LIN {X 0,Y 304.898,Z 957.801,A -85,B 0,C 180,E1 6290.222,E2 6290.222} C_VEL
LIN {X 0,Y 292.236,Z 978.047,A -85,B 0,C 180,E1 6289.106,E2 6289.106} C_VEL
LIN {X 0,Y 278.301,Z 997.321,A -85,B 0,C 180,E1 6287.757,E2 6287.757} C_VEL
LIN {X 0,Y 264.527,Z 1014.363,A -85,B 0,C 180,E1 6286.275,E2 6286.275} C_VEL
LIN {X 0,Y 248.242,Z 1032.202,A -85,B 0,C 180,E1 6284.295,E2 6284.295} C_VEL
LIN {X 0,Y 233.158,Z 1046.985,A -85,B 0,C 180,E1 6282.185,E2 6282.185} C_VEL
LIN {X 0,Y 215.006,Z 1062.935,A -85,B 0,C 180,E1 6279.19,E2 6279.19} C_VEL
LIN {X 0,Y 199.139,Z 1075.414,A -85,B 0,C 180,E1 6276.041,E2 6276.041} C_VEL
LIN {X 0,Y 181.496,Z 1088.037,A -85,B 0,C 180,E1 6271.719,E2 6271.719} C_VEL
LIN {X 0,Y 165.933,Z 1098.063,A -85,B 0,C 180,E1 6266.888,E2 6266.888} C_VEL
LIN {X 0,Y 150.317,Z 1107.482,A -85,B 0,C 180,E1 6260.5,E2 6260.5} C_VEL
LIN {X 0,Y 136.741,Z 1114.997,A -85,B 0,C 180,E1 6252.847,E2 6252.847} C_VEL
LIN {X 0,Y 125.803,Z 1121.052,A -85,B 0,C 180,E1 6243.805,E2 6243.805} C_VEL
LIN {X 0,Y 117.737,Z 1125.633,A -85,B 0,C 180,E1 6232.996,E2 6232.996} C_VEL
LIN {X 0,Y 113.836,Z 1128.278,A -85,B 0,C 180,E1 6223.201,E2 6223.201} C_VEL
LIN {X 0,Y 112.36,Z 1129.83,A -85,B 0,C 180,E1 6213.571,E2 6213.571} C_VEL
LIN {X 0,Y 112.173,Z 1130.41,A -85,B 0,C 180,E1 6205.399,E2 6205.399} C_VEL
LIN {X 0,Y 112.752,Z 1130.33,A -85,B 0,C 180,E1 6196.669,E2 6196.669} C_VEL
LIN {X 0,Y 116.015,Z 1129.028,A -85,B 0,C 180,E1 6184.819,E2 6184.819} C_VEL
LIN {X 0,Y 122.657,Z 1126.25,A -85,B 0,C 180,E1 6174.06,E2 6174.06} C_VEL
LIN {X 0,Y 132.853,Z 1122.064,A -85,B 0,C 180,E1 6164.357,E2 6164.357} C_VEL
LIN {X 0,Y 146.642,Z 1115.907,A -85,B 0,C 180,E1 6155.766,E2 6155.766} C_VEL
LIN {X 0,Y 161.55,Z 1108.77,A -85,B 0,C 180,E1 6149.226,E2 6149.226} C_VEL
LIN {X 0,Y 179.686,Z 1099.063,A -85,B 0,C 180,E1 6143.34,E2 6143.34} C_VEL
LIN {X 0,Y 195.959,Z 1089.416,A -85,B 0,C 180,E1 6139.269,E2 6139.269} C_VEL
LIN {X 0,Y 215.67,Z 1076.309,A -85,B 0,C 180,E1 6135.348,E2 6135.348} C_VEL
LIN {X 0,Y 231.93,Z 1064.205,A -85,B 0,C 180,E1 6132.701,E2 6132.701} C_VEL
LIN {X 0,Y 251.017,Z 1048.279,A -85,B 0,C 180,E1 6130.094,E2 6130.094} C_VEL
LIN {X 0,Y 266.738,Z 1033.492,A -85,B 0,C 180,E1 6128.258,E2 6128.258} C_VEL
LIN {X 0,Y 283.805,Z 1015.52,A -85,B 0,C 180,E1 6126.518,E2 6126.518} C_VEL
LIN {X 0,Y 298.201,Z 998.272,A -85,B 0,C 180,E1 6125.209,E2 6125.209} C_VEL
LIN {X 0,Y 312.738,Z 978.752,A -85,B 0,C 180,E1 6124.022,E2 6124.022} C_VEL
LIN {X 0,Y 325.434,Z 958.993,A -85,B 0,C 180,E1 6123.074,E2 6123.074} C_VEL
LIN {X 0,Y 336.735,Z 939.05,A -85,B 0,C 180,E1 6122.294,E2 6122.294} C_VEL
LIN {X 0,Y 347.411,Z 916.879,A -85,B 0,C 180,E1 6121.59,E2 6121.59} C_VEL
LIN {X 0,Y 355.636,Z 896.806,A -85,B 0,C 180,E1 6121.07,E2 6121.07} C_VEL
LIN {X 0,Y 364.26,Z 871.088,A -85,B 0,C 180,E1 6120.548,E2 6120.548} C_VEL
LIN {X 0,Y 369.901,Z 849.595,A -85,B 0,C 180,E1 6120.212,E2 6120.212} C_VEL
LIN {X 0,Y 374.915,Z 823.874,A -85,B 0,C 180,E1 6119.886,E2 6119.886} C_VEL
LIN {X 0,Y 384.548,Z 747.194,A -85,B 0,C 180,E1 6118.994,E2 6118.994} C_VEL
LIN {X 0,Y 384.545,Z 747.255,A -85,B 0,C 180,E1 6118.358,E2 6118.358} C_VEL
LIN {X 0,Y 374.791,Z 824.894,A -85,B 0,C 180,E1 6117.482,E2 6117.482} C_VEL
LIN {X 0,Y 369.754,Z 850.606,A -85,B 0,C 180,E1 6117.178,E2 6117.178} C_VEL
LIN {X 0,Y 363.934,Z 872.712,A -85,B 0,C 180,E1 6116.896,E2 6116.896} C_VEL
LIN {X 0,Y 355.623,Z 897.463,A -85,B 0,C 180,E1 6116.508,E2 6116.508} C_VEL
LIN {X 0,Y 347.272,Z 917.915,A -85,B 0,C 180,E1 6116.09,E2 6116.09} C_VEL
LIN {X 0,Y 336.01,Z 941.278,A -85,B 0,C 180,E1 6115.48,E2 6115.48} C_VEL
LIN {X 0,Y 324.796,Z 961.093,A -85,B 0,C 180,E1 6114.814,E2 6114.814} C_VEL
LIN {X 0,Y 311.339,Z 982.009,A -85,B 0,C 180,E1 6113.916,E2 6113.916} C_VEL
LIN {X 0,Y 297.261,Z 1000.938,A -85,B 0,C 180,E1 6112.881,E2 6112.881} C_VEL
LIN {X 0,Y 286.778,Z 1013.72,A -85,B 0,C 180,E1 6112.028,E2 6112.028} C_VEL
LIN {X 0,Y 281.639,Z 1019.561,A -85,B 0,C 180,E1 6111.794,E2 6111.794} C_VEL
LIN {X 0,Y 267.373,Z 1033.728,A -85,B 0,C 180,E1 6111.844,E2 6111.844} C_VEL
LIN {X 0,Y 261.888,Z 1038.923,A -85,B 0,C 180,E1 6111.552,E2 6111.552} C_VEL
LIN {X 0,Y 243.935,Z 1055.396,A -85,B 0,C 180,E1 6109.662,E2 6109.662} C_VEL
LIN {X 0,Y 226.368,Z 1069.63,A -85,B 0,C 180,E1 6107.47,E2 6107.47} C_VEL
LIN {X 0,Y 207.429,Z 1083.499,A -85,B 0,C 180,E1 6104.598,E2 6104.598} C_VEL
LIN {X 0,Y 189.12,Z 1095.287,A -85,B 0,C 180,E1 6101.154,E2 6101.154} C_VEL
LIN {X 0,Y 170.844,Z 1106.005,A -85,B 0,C 180,E1 6096.762,E2 6096.762} C_VEL
LIN {X 0,Y 152.99,Z 1115.302,A -85,B 0,C 180,E1 6091.077,E2 6091.077} C_VEL
LIN {X 0,Y 137.723,Z 1122.62,A -85,B 0,C 180,E1 6084.404,E2 6084.404} C_VEL
LIN {X 0,Y 122.504,Z 1129.369,A -85,B 0,C 180,E1 6074.583,E2 6074.583} C_VEL
LIN {X 0,Y 112.831,Z 1133.572,A -85,B 0,C 180,E1 6064.552,E2 6064.552} C_VEL
LIN {X 0,Y 105.971,Z 1136.787,A -85,B 0,C 180,E1 6051.011,E2 6051.011} C_VEL
LIN {X 0,Y 104.147,Z 1137.949,A -85,B 0,C 180,E1 6039.951,E2 6039.951} C_VEL
LIN {X 0,Y 104.146,Z 1138.113,A -85,B 0,C 180,E1 6032.201,E2 6032.201} C_VEL
LIN {X 0,Y 104.106,Z 1137.831,A -85,B 0,C 180,E1 6025.593,E2 6025.593} C_VEL
LIN {X 0,Y 104.641,Z 1136.288,A -85,B 0,C 180,E1 6014.819,E2 6014.819} C_VEL
LIN {X 0,Y 107.92,Z 1133.469,A -85,B 0,C 180,E1 6003.594,E2 6003.594} C_VEL
LIN {X 0,Y 114.969,Z 1129.157,A -85,B 0,C 180,E1 5992.497,E2 5992.497} C_VEL
LIN {X 0,Y 127.083,Z 1122.431,A -85,B 0,C 180,E1 5981.629,E2 5981.629} C_VEL
LIN {X 0,Y 140.009,Z 1115.286,A -85,B 0,C 180,E1 5974.062,E2 5974.062} C_VEL
LIN {X 0,Y 157.991,Z 1104.772,A -85,B 0,C 180,E1 5966.702,E2 5966.702} C_VEL
LIN {X 0,Y 173.714,Z 1094.798,A -85,B 0,C 180,E1 5961.971,E2 5961.971} C_VEL
LIN {X 0,Y 193.113,Z 1081.265,A -85,B 0,C 180,E1 5957.476,E2 5957.476} C_VEL
LIN {X 0,Y 208.714,Z 1069.199,A -85,B 0,C 180,E1 5954.595,E2 5954.595} C_VEL
LIN {X 0,Y 226.805,Z 1053.799,A -85,B 0,C 180,E1 5951.844,E2 5951.844} C_VEL
LIN {X 0,Y 243.473,Z 1037.766,A -85,B 0,C 180,E1 5949.724,E2 5949.724} C_VEL
LIN {X 0,Y 259.698,Z 1020.507,A -85,B 0,C 180,E1 5947.967,E2 5947.967} C_VEL
LIN {X 0,Y 275.239,Z 1001.592,A -85,B 0,C 180,E1 5946.498,E2 5946.498} C_VEL
LIN {X 0,Y 289.714,Z 981.908,A -85,B 0,C 180,E1 5945.311,E2 5945.311} C_VEL
LIN {X 0,Y 302.837,Z 961.222,A -85,B 0,C 180,E1 5944.341,E2 5944.341} C_VEL
LIN {X 0,Y 314.086,Z 941.117,A -85,B 0,C 180,E1 5943.598,E2 5943.598} C_VEL
LIN {X 0,Y 324.895,Z 918.421,A -85,B 0,C 180,E1 5942.943,E2 5942.943} C_VEL
LIN {X 0,Y 333.276,Z 897.7,A -85,B 0,C 180,E1 5942.475,E2 5942.475} C_VEL
LIN {X 0,Y 341.836,Z 871.768,A -85,B 0,C 180,E1 5942.034,E2 5942.034} C_VEL
LIN {X 0,Y 347.498,Z 849.842,A -85,B 0,C 180,E1 5941.734,E2 5941.734} C_VEL
LIN {X 0,Y 352.537,Z 822.943,A -85,B 0,C 180,E1 5941.399,E2 5941.399} C_VEL
LIN {X 0,Y 363.327,Z 734.773,A -85,B 0,C 180,E1 5940.364,E2 5940.364} C_VEL
LIN {X 0,Y 363.314,Z 734.781,A -85,B 0,C 180,E1 5936.149,E2 5936.149} C_VEL
LIN {X 0,Y 352.378,Z 823.667,A -85,B 0,C 180,E1 5935.127,E2 5935.127} C_VEL
LIN {X 0,Y 347.434,Z 849.297,A -85,B 0,C 180,E1 5934.783,E2 5934.783} C_VEL
LIN {X 0,Y 341.984,Z 870.331,A -85,B 0,C 180,E1 5934.432,E2 5934.432} C_VEL
LIN {X 0,Y 333.528,Z 895.974,A -85,B 0,C 180,E1 5933.877,E2 5933.877} C_VEL
LIN {X 0,Y 325.183,Z 916.61,A -85,B 0,C 180,E1 5933.306,E2 5933.306} C_VEL
LIN {X 0,Y 314.045,Z 939.873,A -85,B 0,C 180,E1 5932.499,E2 5932.499} C_VEL
LIN {X 0,Y 303.166,Z 959.23,A -85,B 0,C 180,E1 5931.671,E2 5931.671} C_VEL
LIN {X 0,Y 289.884,Z 979.991,A -85,B 0,C 180,E1 5930.575,E2 5930.575} C_VEL
LIN {X 0,Y 276.242,Z 998.464,A -85,B 0,C 180,E1 5929.337,E2 5929.337} C_VEL
LIN {X 0,Y 260.886,Z 1017.068,A -85,B 0,C 180,E1 5927.779,E2 5927.779} C_VEL
LIN {X 0,Y 244.36,Z 1034.507,A -85,B 0,C 180,E1 5925.878,E2 5925.878} C_VEL
LIN {X 0,Y 227.247,Z 1050.769,A -85,B 0,C 180,E1 5923.578,E2 5923.578} C_VEL
LIN {X 0,Y 209.661,Z 1065.435,A -85,B 0,C 180,E1 5920.784,E2 5920.784} C_VEL
LIN {X 0,Y 191.81,Z 1078.946,A -85,B 0,C 180,E1 5917.323,E2 5917.323} C_VEL
LIN {X 0,Y 173.833,Z 1090.943,A -85,B 0,C 180,E1 5912.973,E2 5912.973} C_VEL
LIN {X 0,Y 156.749,Z 1101.418,A -85,B 0,C 180,E1 5907.599,E2 5907.599} C_VEL
LIN {X 0,Y 140.468,Z 1110.354,A -85,B 0,C 180,E1 5900.689,E2 5900.689} C_VEL
LIN {X 0,Y 126.497,Z 1117.699,A -85,B 0,C 180,E1 5892.213,E2 5892.213} C_VEL
LIN {X 0,Y 115.363,Z 1123.276,A -85,B 0,C 180,E1 5881.853,E2 5881.853} C_VEL
LIN {X 0,Y 108.514,Z 1127.027,A -85,B 0,C 180,E1 5871.061,E2 5871.061} C_VEL
LIN {X 0,Y 104.818,Z 1129.609,A -85,B 0,C 180,E1 5858.227,E2 5858.227} C_VEL
LIN {X 0,Y 104.182,Z 1130.535,A -85,B 0,C 180,E1 5848.9,E2 5848.9} C_VEL
LIN {X 0,Y 104.418,Z 1130.76,A -85,B 0,C 180,E1 5840.075,E2 5840.075} C_VEL
LIN {X 0,Y 106.169,Z 1130.147,A -85,B 0,C 180,E1 5829.607,E2 5829.607} C_VEL
LIN {X 0,Y 110.736,Z 1128.48,A -85,B 0,C 180,E1 5819.024,E2 5819.024} C_VEL
LIN {X 0,Y 120.03,Z 1125.1,A -85,B 0,C 180,E1 5807.564,E2 5807.564} C_VEL
LIN {X 0,Y 132.385,Z 1120.158,A -85,B 0,C 180,E1 5798.233,E2 5798.233} C_VEL
LIN {X 0,Y 148.163,Z 1113.472,A -85,B 0,C 180,E1 5790.252,E2 5790.252} C_VEL
LIN {X 0,Y 165.334,Z 1105.151,A -85,B 0,C 180,E1 5784.047,E2 5784.047} C_VEL
LIN {X 0,Y 183.19,Z 1095.637,A -85,B 0,C 180,E1 5779.217,E2 5779.217} C_VEL
LIN {X 0,Y 202.302,Z 1083.998,A -85,B 0,C 180,E1 5775.186,E2 5775.186} C_VEL
LIN {X 0,Y 219.944,Z 1072.056,A -85,B 0,C 180,E1 5772.199,E2 5772.199} C_VEL
LIN {X 0,Y 238.323,Z 1057.967,A -85,B 0,C 180,E1 5769.615,E2 5769.615} C_VEL
LIN {X 0,Y 254.586,Z 1044.033,A -85,B 0,C 180,E1 5767.674,E2 5767.674} C_VEL
LIN {X 0,Y 273.346,Z 1025.88,A -85,B 0,C 180,E1 5765.748,E2 5765.748} C_VEL
LIN {X 0,Y 287.836,Z 1010.027,A -85,B 0,C 180,E1 5764.446,E2 5764.446} C_VEL
LIN {X 0,Y 303.927,Z 990.158,A -85,B 0,C 180,E1 5763.148,E2 5763.148} C_VEL
LIN {X 0,Y 316.703,Z 972.103,A -85,B 0,C 180,E1 5762.214,E2 5762.214} C_VEL
LIN {X 0,Y 329.558,Z 951.587,A -85,B 0,C 180,E1 5761.354,E2 5761.354} C_VEL
LIN {X 0,Y 340.985,Z 930.062,A -85,B 0,C 180,E1 5760.627,E2 5760.627} C_VEL
LIN {X 0,Y 351.289,Z 907.567,A -85,B 0,C 180,E1 5760.02,E2 5760.02} C_VEL
LIN {X 0,Y 359.524,Z 885.529,A -85,B 0,C 180,E1 5759.548,E2 5759.548} C_VEL
LIN {X 0,Y 366.123,Z 864.196,A -85,B 0,C 180,E1 5759.173,E2 5759.173} C_VEL
LIN {X 0,Y 372.227,Z 838.404,A -85,B 0,C 180,E1 5758.823,E2 5758.823} C_VEL
LIN {X 0,Y 374.389,Z 826.988,A -85,B 0,C 180,E1 5758.686,E2 5758.686} C_VEL
LIN {X 0,Y 369.323,Z 851.712,A -85,B 0,C 180,E1 5758.408,E2 5758.408} C_VEL
LIN {X 0,Y 362.984,Z 875.26,A -85,B 0,C 180,E1 5758.127,E2 5758.127} C_VEL
LIN {X 0,Y 354.73,Z 898.996,A -85,B 0,C 180,E1 5757.776,E2 5757.776} C_VEL
LIN {X 0,Y 346.324,Z 919.231,A -85,B 0,C 180,E1 5757.388,E2 5757.388} C_VEL
LIN {X 0,Y 334.979,Z 942.269,A -85,B 0,C 180,E1 5756.825,E2 5756.825} C_VEL
LIN {X 0,Y 324.166,Z 961.147,A -85,B 0,C 180,E1 5756.233,E2 5756.233} C_VEL
LIN {X 0,Y 310.959,Z 981.492,A -85,B 0,C 180,E1 5755.424,E2 5755.424} C_VEL
LIN {X 0,Y 296.365,Z 1000.906,A -85,B 0,C 180,E1 5754.437,E2 5754.437} C_VEL
LIN {X 0,Y 280.919,Z 1019.268,A -85,B 0,C 180,E1 5753.248,E2 5753.248} C_VEL
LIN {X 0,Y 264.666,Z 1036.202,A -85,B 0,C 180,E1 5751.819,E2 5751.819} C_VEL
LIN {X 0,Y 261.888,Z 1038.923,A -85,B 0,C 180,E1 5751.552,E2 5751.552} C_VEL
LIN {X 0,Y 256.284,Z 1044.179,A -85,B 0,C 180,E1 5751.234,E2 5751.234} C_VEL
LIN {X 0,Y 240.739,Z 1056.943,A -85,B 0,C 180,E1 5751.117,E2 5751.117} C_VEL
LIN {X 0,Y 234.837,Z 1061.634,A -85,B 0,C 180,E1 5750.725,E2 5750.725} C_VEL
LIN {X 0,Y 214.477,Z 1076.988,A -85,B 0,C 180,E1 5748.163,E2 5748.163} C_VEL
LIN {X 0,Y 196.365,Z 1089.127,A -85,B 0,C 180,E1 5745.349,E2 5745.349} C_VEL
LIN {X 0,Y 175.347,Z 1101.608,A -85,B 0,C 180,E1 5741.19,E2 5741.19} C_VEL
LIN {X 0,Y 157.901,Z 1110.829,A -85,B 0,C 180,E1 5736.665,E2 5736.665} C_VEL
LIN {X 0,Y 138.008,Z 1120.207,A -85,B 0,C 180,E1 5729.562,E2 5729.562} C_VEL
LIN {X 0,Y 123.227,Z 1126.513,A -85,B 0,C 180,E1 5721.914,E2 5721.914} C_VEL
LIN {X 0,Y 108.995,Z 1132.188,A -85,B 0,C 180,E1 5710.41,E2 5710.41} C_VEL
LIN {X 0,Y 100.988,Z 1135.372,A -85,B 0,C 180,E1 5699.023,E2 5699.023} C_VEL
LIN {X 0,Y 96.601,Z 1137.46,A -85,B 0,C 180,E1 5684.997,E2 5684.997} C_VEL
LIN {X 0,Y 96.105,Z 1137.881,A -85,B 0,C 180,E1 5674.177,E2 5674.177} C_VEL
LIN {X 0,Y 96.151,Z 1137.648,A -85,B 0,C 180,E1 5667.616,E2 5667.616} C_VEL
LIN {X 0,Y 96.272,Z 1136.668,A -85,B 0,C 180,E1 5658.011,E2 5658.011} C_VEL
LIN {X 0,Y 99.377,Z 1133.984,A -85,B 0,C 180,E1 5644.364,E2 5644.364} C_VEL
LIN {X 0,Y 106.402,Z 1129.901,A -85,B 0,C 180,E1 5632.351,E2 5632.351} C_VEL
LIN {X 0,Y 117.811,Z 1124.128,A -85,B 0,C 180,E1 5621.453,E2 5621.453} C_VEL
LIN {X 0,Y 132.74,Z 1116.376,A -85,B 0,C 180,E1 5612.47,E2 5612.47} C_VEL
LIN {X 0,Y 148.831,Z 1107.645,A -85,B 0,C 180,E1 5605.808,E2 5605.808} C_VEL
LIN {X 0,Y 167.328,Z 1096.567,A -85,B 0,C 180,E1 5600.252,E2 5600.252} C_VEL
LIN {X 0,Y 184.427,Z 1085.333,A -85,B 0,C 180,E1 5596.336,E2 5596.336} C_VEL
LIN {X 0,Y 204.05,Z 1070.901,A -85,B 0,C 180,E1 5592.8,E2 5592.8} C_VEL
LIN {X 0,Y 220.592,Z 1057.353,A -85,B 0,C 180,E1 5590.387,E2 5590.387} C_VEL
LIN {X 0,Y 239.369,Z 1040.102,A -85,B 0,C 180,E1 5588.11,E2 5588.11} C_VEL
LIN {X 0,Y 254.642,Z 1024.339,A -85,B 0,C 180,E1 5586.539,E2 5586.539} C_VEL
LIN {X 0,Y 271.519,Z 1004.747,A -85,B 0,C 180,E1 5585.033,E2 5585.033} C_VEL
LIN {X 0,Y 285.157,Z 986.751,A -85,B 0,C 180,E1 5583.977,E2 5583.977} C_VEL
LIN {X 0,Y 299.377,Z 965.518,A -85,B 0,C 180,E1 5582.993,E2 5582.993} C_VEL
LIN {X 0,Y 310.638,Z 946.051,A -85,B 0,C 180,E1 5582.29,E2 5582.29} C_VEL
LIN {X 0,Y 321.402,Z 924.816,A -85,B 0,C 180,E1 5581.679,E2 5581.679} C_VEL
LIN {X 0,Y 331.035,Z 902.056,A -85,B 0,C 180,E1 5581.178,E2 5581.178} C_VEL
LIN {X 0,Y 338.724,Z 880.402,A -85,B 0,C 180,E1 5580.816,E2 5580.816} C_VEL
LIN {X 0,Y 345.88,Z 854.864,A -85,B 0,C 180,E1 5580.476,E2 5580.476} C_VEL
LIN {X 0,Y 350.591,Z 832.594,A -85,B 0,C 180,E1 5580.208,E2 5580.208} C_VEL
LIN {X 0,Y 355.236,Z 799.743,A -85,B 0,C 180,E1 5579.838,E2 5579.838} C_VEL
LIN {X 0,Y 362.17,Z 742.553,A -85,B 0,C 180,E1 5579.169,E2 5579.169} C_VEL
LIN {X 0,Y 362.139,Z 742.775,A -85,B 0,C 180,E1 5577.324,E2 5577.324} C_VEL
LIN {X 0,Y 351.964,Z 824.217,A -85,B 0,C 180,E1 5576.424,E2 5576.424} C_VEL
LIN {X 0,Y 346.986,Z 849.69,A -85,B 0,C 180,E1 5576.1,E2 5576.1} C_VEL
LIN {X 0,Y 341.458,Z 870.814,A -85,B 0,C 180,E1 5575.769,E2 5575.769} C_VEL
LIN {X 0,Y 333.105,Z 895.936,A -85,B 0,C 180,E1 5575.26,E2 5575.26} C_VEL
LIN {X 0,Y 324.837,Z 916.256,A -85,B 0,C 180,E1 5574.734,E2 5574.734} C_VEL
LIN {X 0,Y 314.178,Z 938.565,A -85,B 0,C 180,E1 5574.019,E2 5574.019} C_VEL
LIN {X 0,Y 303.074,Z 958.259,A -85,B 0,C 180,E1 5573.242,E2 5573.242} C_VEL
LIN {X 0,Y 290.115,Z 978.517,A -85,B 0,C 180,E1 5572.259,E2 5572.259} C_VEL
LIN {X 0,Y 275.818,Z 997.811,A -85,B 0,C 180,E1 5571.066,E2 5571.066} C_VEL
LIN {X 0,Y 261.649,Z 1014.862,A -85,B 0,C 180,E1 5569.75,E2 5569.75} C_VEL
LIN {X 0,Y 244.372,Z 1033.172,A -85,B 0,C 180,E1 5567.936,E2 5567.936} C_VEL
LIN {X 0,Y 228.735,Z 1047.924,A -85,B 0,C 180,E1 5566.038,E2 5566.038} C_VEL
LIN {X 0,Y 209.802,Z 1063.815,A -85,B 0,C 180,E1 5563.325,E2 5563.325} C_VEL
LIN {X 0,Y 193.125,Z 1076.269,A -85,B 0,C 180,E1 5560.441,E2 5560.441} C_VEL
LIN {X 0,Y 173.544,Z 1089.357,A -85,B 0,C 180,E1 5556.214,E2 5556.214} C_VEL
LIN {X 0,Y 156.874,Z 1099.288,A -85,B 0,C 180,E1 5551.594,E2 5551.594} C_VEL
LIN {X 0,Y 139.137,Z 1108.901,A -85,B 0,C 180,E1 5545.01,E2 5545.01} C_VEL
LIN {X 0,Y 124.722,Z 1116,A -85,B 0,C 180,E1 5537.524,E2 5537.524} C_VEL
LIN {X 0,Y 111.756,Z 1122.197,A -85,B 0,C 180,E1 5527.474,E2 5527.474} C_VEL
LIN {X 0,Y 102.46,Z 1126.582,A -85,B 0,C 180,E1 5515.429,E2 5515.429} C_VEL
LIN {X 0,Y 97.809,Z 1129.224,A -85,B 0,C 180,E1 5503.599,E2 5503.599} C_VEL
LIN {X 0,Y 96.26,Z 1130.736,A -85,B 0,C 180,E1 5491.19,E2 5491.19} C_VEL
LIN {X 0,Y 96.307,Z 1131.112,A -85,B 0,C 180,E1 5481.642,E2 5481.642} C_VEL
LIN {X 0,Y 98.214,Z 1130.547,A -85,B 0,C 180,E1 5469.125,E2 5469.125} C_VEL
LIN {X 0,Y 103.431,Z 1128.854,A -85,B 0,C 180,E1 5457.223,E2 5457.223} C_VEL
LIN {X 0,Y 113.543,Z 1125.542,A -85,B 0,C 180,E1 5445.21,E2 5445.21} C_VEL
LIN {X 0,Y 127.407,Z 1120.397,A -85,B 0,C 180,E1 5435.294,E2 5435.294} C_VEL
LIN {X 0,Y 144.15,Z 1113.695,A -85,B 0,C 180,E1 5427.393,E2 5427.393} C_VEL
LIN {X 0,Y 162.276,Z 1105.281,A -85,B 0,C 180,E1 5421.318,E2 5421.318} C_VEL
LIN {X 0,Y 180.625,Z 1095.831,A -85,B 0,C 180,E1 5416.727,E2 5416.727} C_VEL
LIN {X 0,Y 200.056,Z 1084.314,A -85,B 0,C 180,E1 5412.934,E2 5412.934} C_VEL
LIN {X 0,Y 218.345,Z 1072.212,A -85,B 0,C 180,E1 5410.075,E2 5410.075} C_VEL
LIN {X 0,Y 237.083,Z 1058.092,A -85,B 0,C 180,E1 5407.646,E2 5407.646} C_VEL
LIN {X 0,Y 254.259,Z 1043.579,A -85,B 0,C 180,E1 5405.764,E2 5405.764} C_VEL
LIN {X 0,Y 272.646,Z 1025.952,A -85,B 0,C 180,E1 5404.03,E2 5404.03} C_VEL
LIN {X 0,Y 287.652,Z 1009.7,A -85,B 0,C 180,E1 5402.789,E2 5402.789} C_VEL
LIN {X 0,Y 304.578,Z 988.822,A -85,B 0,C 180,E1 5401.536,E2 5401.536} C_VEL
LIN {X 0,Y 316.991,Z 971.339,A -85,B 0,C 180,E1 5400.708,E2 5400.708} C_VEL
LIN {X 0,Y 330.466,Z 949.685,A -85,B 0,C 180,E1 5399.88,E2 5399.88} C_VEL
LIN {X 0,Y 340.993,Z 929.917,A -85,B 0,C 180,E1 5399.263,E2 5399.263} C_VEL
LIN {X 0,Y 348.65,Z 913.526,A -85,B 0,C 180,E1 5398.829,E2 5398.829} C_VEL
LIN {X 0,Y 339.095,Z 933.848,A -85,B 0,C 180,E1 5398.412,E2 5398.412} C_VEL
LIN {X 0,Y 326.21,Z 957.146,A -85,B 0,C 180,E1 5397.784,E2 5397.784} C_VEL
LIN {X 0,Y 314.851,Z 974.953,A -85,B 0,C 180,E1 5397.169,E2 5397.169} C_VEL
LIN {X 0,Y 300.164,Z 995.311,A -85,B 0,C 180,E1 5396.289,E2 5396.289} C_VEL
LIN {X 0,Y 284.942,Z 1013.651,A -85,B 0,C 180,E1 5395.268,E2 5395.268} C_VEL
LIN {X 0,Y 268.45,Z 1031.443,A -85,B 0,C 180,E1 5393.985,E2 5393.985} C_VEL
LIN {X 0,Y 251.158,Z 1047.749,A -85,B 0,C 180,E1 5392.439,E2 5392.439} C_VEL
LIN {X 0,Y 234.837,Z 1061.634,A -85,B 0,C 180,E1 5390.725,E2 5390.725} C_VEL
LIN {X 0,Y 228.832,Z 1066.279,A -85,B 0,C 180,E1 5390.299,E2 5390.299} C_VEL
LIN {X 0,Y 212.174,Z 1077.499,A -85,B 0,C 180,E1 5389.942,E2 5389.942} C_VEL
LIN {X 0,Y 205.939,Z 1081.635,A -85,B 0,C 180,E1 5389.4,E2 5389.4} C_VEL
LIN {X 0,Y 185.343,Z 1094.397,A -85,B 0,C 180,E1 5386.185,E2 5386.185} C_VEL
LIN {X 0,Y 166.74,Z 1104.677,A -85,B 0,C 180,E1 5382.455,E2 5382.455} C_VEL
LIN {X 0,Y 146.562,Z 1114.471,A -85,B 0,C 180,E1 5377.075,E2 5377.075} C_VEL
LIN {X 0,Y 130.25,Z 1121.534,A -85,B 0,C 180,E1 5371.063,E2 5371.063} C_VEL
LIN {X 0,Y 112.545,Z 1128.435,A -85,B 0,C 180,E1 5361.428,E2 5361.428} C_VEL
LIN {X 0,Y 100.493,Z 1132.754,A -85,B 0,C 180,E1 5350.871,E2 5350.871} C_VEL
LIN {X 0,Y 91.508,Z 1136.032,A -85,B 0,C 180,E1 5336.363,E2 5336.363} C_VEL
LIN {X 0,Y 88.303,Z 1137.353,A -85,B 0,C 180,E1 5322.424,E2 5322.424} C_VEL
LIN {X 0,Y 88.146,Z 1137.533,A -85,B 0,C 180,E1 5312.601,E2 5312.601} C_VEL
LIN {X 0,Y 88.11,Z 1137.285,A -85,B 0,C 180,E1 5305.444,E2 5305.444} C_VEL
LIN {X 0,Y 88.864,Z 1135.831,A -85,B 0,C 180,E1 5292.989,E2 5292.989} C_VEL
LIN {X 0,Y 93.482,Z 1132.818,A -85,B 0,C 180,E1 5279.109,E2 5279.109} C_VEL
LIN {X 0,Y 102.344,Z 1128.482,A -85,B 0,C 180,E1 5266.851,E2 5266.851} C_VEL
LIN {X 0,Y 116.715,Z 1121.713,A -85,B 0,C 180,E1 5255.524,E2 5255.524} C_VEL
LIN {X 0,Y 131.413,Z 1114.545,A -85,B 0,C 180,E1 5248.04,E2 5248.04} C_VEL
LIN {X 0,Y 151.114,Z 1104.06,A -85,B 0,C 180,E1 5241.097,E2 5241.097} C_VEL
LIN {X 0,Y 168.096,Z 1094.047,A -85,B 0,C 180,E1 5236.728,E2 5236.728} C_VEL
LIN {X 0,Y 188.593,Z 1080.544,A -85,B 0,C 180,E1 5232.697,E2 5232.697} C_VEL
LIN {X 0,Y 205.228,Z 1068.259,A -85,B 0,C 180,E1 5230.102,E2 5230.102} C_VEL
LIN {X 0,Y 224.052,Z 1052.798,A -85,B 0,C 180,E1 5227.694,E2 5227.694} C_VEL
LIN {X 0,Y 240.272,Z 1037.725,A -85,B 0,C 180,E1 5225.955,E2 5225.955} C_VEL
LIN {X 0,Y 257.233,Z 1020.236,A -85,B 0,C 180,E1 5224.404,E2 5224.404} C_VEL
LIN {X 0,Y 273.001,Z 1001.58,A -85,B 0,C 180,E1 5223.149,E2 5223.149} C_VEL
LIN {X 0,Y 287.176,Z 982.789,A -85,B 0,C 180,E1 5222.171,E2 5222.171} C_VEL
LIN {X 0,Y 301.047,Z 961.594,A -85,B 0,C 180,E1 5221.31,E2 5221.31} C_VEL
LIN {X 0,Y 311.991,Z 942.505,A -85,B 0,C 180,E1 5220.705,E2 5220.705} C_VEL
LIN {X 0,Y 323.467,Z 919.17,A -85,B 0,C 180,E1 5220.127,E2 5220.127} C_VEL
LIN {X 0,Y 331.969,Z 898.63,A -85,B 0,C 180,E1 5219.732,E2 5219.732} C_VEL
LIN {X 0,Y 340.36,Z 874.209,A -85,B 0,C 180,E1 5219.377,E2 5219.377} C_VEL
LIN {X 0,Y 346.449,Z 851.423,A -85,B 0,C 180,E1 5219.109,E2 5219.109} C_VEL
LIN {X 0,Y 351.487,Z 826.523,A -85,B 0,C 180,E1 5218.831,E2 5218.831} C_VEL
LIN {X 0,Y 358.252,Z 774.063,A -85,B 0,C 180,E1 5218.263,E2 5218.263} C_VEL
LIN {X 0,Y 351.418,Z 826.92,A -85,B 0,C 180,E1 5217.7,E2 5217.7} C_VEL
LIN {X 0,Y 346.411,Z 851.383,A -85,B 0,C 180,E1 5217.402,E2 5217.402} C_VEL
LIN {X 0,Y 340.564,Z 873.224,A -85,B 0,C 180,E1 5217.075,E2 5217.075} C_VEL
LIN {X 0,Y 332.542,Z 896.764,A -85,B 0,C 180,E1 5216.626,E2 5216.626} C_VEL
LIN {X 0,Y 324.203,Z 917.019,A -85,B 0,C 180,E1 5216.136,E2 5216.136} C_VEL
LIN {X 0,Y 312.958,Z 940.12,A -85,B 0,C 180,E1 5215.44,E2 5215.44} C_VEL
LIN {X 0,Y 301.752,Z 959.688,A -85,B 0,C 180,E1 5214.714,E2 5214.714} C_VEL
LIN {X 0,Y 288.177,Z 980.471,A -85,B 0,C 180,E1 5213.76,E2 5213.76} C_VEL
LIN {X 0,Y 273.963,Z 999.258,A -85,B 0,C 180,E1 5212.661,E2 5212.661} C_VEL
LIN {X 0,Y 258.515,Z 1017.48,A -85,B 0,C 180,E1 5211.324,E2 5211.324} C_VEL
LIN {X 0,Y 241.875,Z 1034.566,A -85,B 0,C 180,E1 5209.698,E2 5209.698} C_VEL
LIN {X 0,Y 225.068,Z 1050.052,A -85,B 0,C 180,E1 5207.791,E2 5207.791} C_VEL
LIN {X 0,Y 206.716,Z 1064.94,A -85,B 0,C 180,E1 5205.332,E2 5205.332} C_VEL
LIN {X 0,Y 189.68,Z 1077.315,A -85,B 0,C 180,E1 5202.581,E2 5202.581} C_VEL
LIN {X 0,Y 169.736,Z 1090.17,A -85,B 0,C 180,E1 5198.553,E2 5198.553} C_VEL
LIN {X 0,Y 153.178,Z 1099.677,A -85,B 0,C 180,E1 5194.266,E2 5194.266} C_VEL
LIN {X 0,Y 134.645,Z 1109.267,A -85,B 0,C 180,E1 5187.842,E2 5187.842} C_VEL
LIN {X 0,Y 119.392,Z 1116.355,A -85,B 0,C 180,E1 5180.398,E2 5180.398} C_VEL
LIN {X 0,Y 105.443,Z 1122.531,A -85,B 0,C 180,E1 5170.153,E2 5170.153} C_VEL
LIN {X 0,Y 95.577,Z 1126.751,A -85,B 0,C 180,E1 5158.085,E2 5158.085} C_VEL
LIN {X 0,Y 90.188,Z 1129.426,A -85,B 0,C 180,E1 5145.431,E2 5145.431} C_VEL
LIN {X 0,Y 88.306,Z 1130.927,A -85,B 0,C 180,E1 5132.596,E2 5132.596} C_VEL
LIN {X 0,Y 88.286,Z 1131.356,A -85,B 0,C 180,E1 5122.189,E2 5122.189} C_VEL
LIN {X 0,Y 90.097,Z 1131.009,A -85,B 0,C 180,E1 5109.198,E2 5109.198} C_VEL
LIN {X 0,Y 95.88,Z 1129.335,A -85,B 0,C 180,E1 5095.726,E2 5095.726} C_VEL
LIN {X 0,Y 105.665,Z 1126.417,A -85,B 0,C 180,E1 5084.013,E2 5084.013} C_VEL
LIN {X 0,Y 121.216,Z 1121.207,A -85,B 0,C 180,E1 5072.985,E2 5072.985} C_VEL
LIN {X 0,Y 136.643,Z 1115.408,A -85,B 0,C 180,E1 5065.834,E2 5065.834} C_VEL
LIN {X 0,Y 156.753,Z 1106.756,A -85,B 0,C 180,E1 5059.254,E2 5059.254} C_VEL
LIN {X 0,Y 173.979,Z 1098.287,A -85,B 0,C 180,E1 5055.087,E2 5055.087} C_VEL
LIN {X 0,Y 194.686,Z 1086.753,A -85,B 0,C 180,E1 5051.197,E2 5051.197} C_VEL
LIN {X 0,Y 212.337,Z 1075.516,A -85,B 0,C 180,E1 5048.548,E2 5048.548} C_VEL
LIN {X 0,Y 231.328,Z 1062.035,A -85,B 0,C 180,E1 5046.197,E2 5046.197} C_VEL
LIN {X 0,Y 249.67,Z 1047.054,A -85,B 0,C 180,E1 5044.28,E2 5044.28} C_VEL
LIN {X 0,Y 266.289,Z 1031.92,A -85,B 0,C 180,E1 5042.794,E2 5042.794} C_VEL
LIN {X 0,Y 283.882,Z 1013.647,A -85,B 0,C 180,E1 5041.413,E2 5041.413} C_VEL
LIN {X 0,Y 297.977,Z 997.138,A -85,B 0,C 180,E1 5040.426,E2 5040.426} C_VEL
LIN {X 0,Y 313.984,Z 975.725,A -85,B 0,C 180,E1 5039.413,E2 5039.413} C_VEL
LIN {X 0,Y 321.35,Z 964.773,A -85,B 0,C 180,E1 5038.986,E2 5038.986} C_VEL
LIN {X 0,Y 307.111,Z 985.487,A -85,B 0,C 180,E1 5038.249,E2 5038.249} C_VEL
LIN {X 0,Y 293.259,Z 1003.278,A -85,B 0,C 180,E1 5037.455,E2 5037.455} C_VEL
LIN {X 0,Y 275.547,Z 1023.238,A -85,B 0,C 180,E1 5036.295,E2 5036.295} C_VEL
LIN {X 0,Y 259.918,Z 1038.802,A -85,B 0,C 180,E1 5035.113,E2 5035.113} C_VEL
LIN {X 0,Y 240.568,Z 1055.916,A -85,B 0,C 180,E1 5033.403,E2 5033.403} C_VEL
LIN {X 0,Y 223.376,Z 1069.343,A -85,B 0,C 180,E1 5031.595,E2 5031.595} C_VEL
LIN {X 0,Y 205.939,Z 1081.635,A -85,B 0,C 180,E1 5029.4,E2 5029.4} C_VEL
LIN {X 0,Y 199.639,Z 1085.668,A -85,B 0,C 180,E1 5028.81,E2 5028.81} C_VEL
LIN {X 0,Y 181.135,Z 1095.771,A -85,B 0,C 180,E1 5028.027,E2 5028.027} C_VEL
LIN {X 0,Y 175.564,Z 1098.727,A -85,B 0,C 180,E1 5027.344,E2 5027.344} C_VEL
LIN {X 0,Y 155.029,Z 1109.02,A -85,B 0,C 180,E1 5023.128,E2 5023.128} C_VEL
LIN {X 0,Y 135.232,Z 1117.863,A -85,B 0,C 180,E1 5017.554,E2 5017.554} C_VEL
LIN {X 0,Y 116.623,Z 1124.977,A -85,B 0,C 180,E1 5009.991,E2 5009.991} C_VEL
LIN {X 0,Y 100.642,Z 1130.555,A -85,B 0,C 180,E1 4999.908,E2 4999.908} C_VEL
LIN {X 0,Y 88.392,Z 1134.386,A -85,B 0,C 180,E1 4986.568,E2 4986.568} C_VEL
LIN {X 0,Y 82.153,Z 1136.413,A -85,B 0,C 180,E1 4972.922,E2 4972.922} C_VEL
LIN {X 0,Y 80.09,Z 1137.299,A -85,B 0,C 180,E1 4957.893,E2 4957.893} C_VEL
LIN {X 0,Y 80.192,Z 1137.14,A -85,B 0,C 180,E1 4949.286,E2 4949.286} C_VEL
LIN {X 0,Y 80.155,Z 1136.502,A -85,B 0,C 180,E1 4939.942,E2 4939.942} C_VEL
LIN {X 0,Y 82.111,Z 1134.794,A -85,B 0,C 180,E1 4927.066,E2 4927.066} C_VEL
LIN {X 0,Y 88.82,Z 1131.48,A -85,B 0,C 180,E1 4912.562,E2 4912.562} C_VEL
LIN {X 0,Y 101.641,Z 1125.897,A -85,B 0,C 180,E1 4898.998,E2 4898.998} C_VEL
LIN {X 0,Y 115.85,Z 1119.686,A -85,B 0,C 180,E1 4890.039,E2 4890.039} C_VEL
LIN {X 0,Y 134.919,Z 1110.639,A -85,B 0,C 180,E1 4882.122,E2 4882.122} C_VEL
LIN {X 0,Y 151.77,Z 1101.777,A -85,B 0,C 180,E1 4877.197,E2 4877.197} C_VEL
LIN {X 0,Y 172.221,Z 1089.783,A -85,B 0,C 180,E1 4872.738,E2 4872.738} C_VEL
LIN {X 0,Y 190.676,Z 1077.513,A -85,B 0,C 180,E1 4869.645,E2 4869.645} C_VEL
LIN {X 0,Y 209.589,Z 1063.509,A -85,B 0,C 180,E1 4867.108,E2 4867.108} C_VEL
LIN {X 0,Y 226.908,Z 1048.926,A -85,B 0,C 180,E1 4865.194,E2 4865.194} C_VEL
LIN {X 0,Y 243.469,Z 1033.464,A -85,B 0,C 180,E1 4863.652,E2 4863.652} C_VEL
LIN {X 0,Y 260.55,Z 1015.372,A -85,B 0,C 180,E1 4862.284,E2 4862.284} C_VEL
LIN {X 0,Y 274.543,Z 998.703,A -85,B 0,C 180,E1 4861.308,E2 4861.308} C_VEL
LIN {X 0,Y 290.475,Z 977.15,A -85,B 0,C 180,E1 4860.337,E2 4860.337} C_VEL
LIN {X 0,Y 302.473,Z 958.495,A -85,B 0,C 180,E1 4859.678,E2 4859.678} C_VEL
LIN {X 0,Y 315.009,Z 936.182,A -85,B 0,C 180,E1 4859.067,E2 4859.067} C_VEL
LIN {X 0,Y 325.06,Z 914.975,A -85,B 0,C 180,E1 4858.626,E2 4858.626} C_VEL
LIN {X 0,Y 334.395,Z 891.859,A -85,B 0,C 180,E1 4858.254,E2 4858.254} C_VEL
LIN {X 0,Y 335.986,Z 887.146,A -85,B 0,C 180,E1 4858.191,E2 4858.191} C_VEL
LIN {X 0,Y 326.73,Z 911.076,A -85,B 0,C 180,E1 4857.699,E2 4857.699} C_VEL
LIN {X 0,Y 317.349,Z 931.239,A -85,B 0,C 180,E1 4857.187,E2 4857.187} C_VEL
LIN {X 0,Y 305.54,Z 953.112,A -85,B 0,C 180,E1 4856.496,E2 4856.496} C_VEL
LIN {X 0,Y 292.791,Z 973.192,A -85,B 0,C 180,E1 4855.707,E2 4855.707} C_VEL
LIN {X 0,Y 278.647,Z 992.885,A -85,B 0,C 180,E1 4854.734,E2 4854.734} C_VEL
LIN {X 0,Y 263.351,Z 1011.288,A -85,B 0,C 180,E1 4853.579,E2 4853.579} C_VEL
LIN {X 0,Y 248.217,Z 1027.568,A -85,B 0,C 180,E1 4852.292,E2 4852.292} C_VEL
LIN {X 0,Y 230.113,Z 1044.708,A -85,B 0,C 180,E1 4850.529,E2 4850.529} C_VEL
LIN {X 0,Y 213.777,Z 1058.461,A -85,B 0,C 180,E1 4848.671,E2 4848.671} C_VEL
LIN {X 0,Y 192.871,Z 1074.008,A -85,B 0,C 180,E1 4845.804,E2 4845.804} C_VEL
LIN {X 0,Y 175.749,Z 1085.246,A -85,B 0,C 180,E1 4842.903,E2 4842.903} C_VEL
LIN {X 0,Y 154.884,Z 1097.384,A -85,B 0,C 180,E1 4838.378,E2 4838.378} C_VEL
LIN {X 0,Y 137.567,Z 1106.253,A -85,B 0,C 180,E1 4833.382,E2 4833.382} C_VEL
LIN {X 0,Y 118.6,Z 1114.95,A -85,B 0,C 180,E1 4825.713,E2 4825.713} C_VEL
LIN {X 0,Y 104.03,Z 1120.954,A -85,B 0,C 180,E1 4816.927,E2 4816.927} C_VEL
LIN {X 0,Y 91.404,Z 1126.005,A -85,B 0,C 180,E1 4804.67,E2 4804.67} C_VEL
LIN {X 0,Y 83.561,Z 1129.194,A -85,B 0,C 180,E1 4790.305,E2 4790.305} C_VEL
LIN {X 0,Y 80.632,Z 1130.832,A -85,B 0,C 180,E1 4777.123,E2 4777.123} C_VEL
LIN {X 0,Y 80.182,Z 1131.45,A -85,B 0,C 180,E1 4767.141,E2 4767.141} C_VEL
LIN {X 0,Y 80.718,Z 1131.59,A -85,B 0,C 180,E1 4756.387,E2 4756.387} C_VEL
LIN {X 0,Y 83.89,Z 1130.912,A -85,B 0,C 180,E1 4743.068,E2 4743.068} C_VEL
LIN {X 0,Y 91.326,Z 1129.071,A -85,B 0,C 180,E1 4729.761,E2 4729.761} C_VEL
LIN {X 0,Y 105.548,Z 1125.05,A -85,B 0,C 180,E1 4716.367,E2 4716.367} C_VEL
LIN {X 0,Y 120.064,Z 1120.381,A -85,B 0,C 180,E1 4708.021,E2 4708.021} C_VEL
LIN {X 0,Y 139.758,Z 1113.099,A -85,B 0,C 180,E1 4700.407,E2 4700.407} C_VEL
LIN {X 0,Y 157.707,Z 1105.37,A -85,B 0,C 180,E1 4695.483,E2 4695.483} C_VEL
LIN {X 0,Y 178.391,Z 1095.229,A -85,B 0,C 180,E1 4691.219,E2 4691.219} C_VEL
LIN {X 0,Y 197.568,Z 1084.315,A -85,B 0,C 180,E1 4688.147,E2 4688.147} C_VEL
LIN {X 0,Y 217.991,Z 1071.224,A -85,B 0,C 180,E1 4685.528,E2 4685.528} C_VEL
LIN {X 0,Y 236.433,Z 1057.577,A -85,B 0,C 180,E1 4683.567,E2 4683.567} C_VEL
LIN {X 0,Y 254.124,Z 1042.955,A -85,B 0,C 180,E1 4681.973,E2 4681.973} C_VEL
LIN {X 0,Y 271.985,Z 1026.095,A -85,B 0,C 180,E1 4680.578,E2 4680.578} C_VEL
LIN {X 0,Y 286.979,Z 1010.179,A -85,B 0,C 180,E1 4679.546,E2 4679.546} C_VEL
LIN {X 0,Y 294.006,Z 1002.03,A -85,B 0,C 180,E1 4679.094,E2 4679.094} C_VEL
LIN {X 0,Y 276.626,Z 1021.637,A -85,B 0,C 180,E1 4678.082,E2 4678.082} C_VEL
LIN {X 0,Y 261.317,Z 1036.848,A -85,B 0,C 180,E1 4677.057,E2 4677.057} C_VEL
LIN {X 0,Y 242.689,Z 1053.458,A -85,B 0,C 180,E1 4675.602,E2 4675.602} C_VEL
LIN {X 0,Y 223.286,Z 1068.494,A -85,B 0,C 180,E1 4673.794,E2 4673.794} C_VEL
LIN {X 0,Y 203.213,Z 1082.398,A -85,B 0,C 180,E1 4671.497,E2 4671.497} C_VEL
LIN {X 0,Y 182.62,Z 1094.734,A -85,B 0,C 180,E1 4668.544,E2 4668.544} C_VEL
LIN {X 0,Y 175.564,Z 1098.727,A -85,B 0,C 180,E1 4667.344,E2 4667.344} C_VEL
LIN {X 0,Y 169.002,Z 1102.063,A -85,B 0,C 180,E1 4666.515,E2 4666.515} C_VEL
LIN {X 0,Y 150.843,Z 1109.987,A -85,B 0,C 180,E1 4665.228,E2 4665.228} C_VEL
LIN {X 0,Y 144.165,Z 1112.705,A -85,B 0,C 180,E1 4664.112,E2 4664.112} C_VEL
LIN {X 0,Y 125.554,Z 1120.138,A -85,B 0,C 180,E1 4658.713,E2 4658.713} C_VEL
LIN {X 0,Y 106.66,Z 1126.84,A -85,B 0,C 180,E1 4650.673,E2 4650.673} C_VEL
LIN {X 0,Y 89.957,Z 1131.856,A -85,B 0,C 180,E1 4639.099,E2 4639.099} C_VEL
LIN {X 0,Y 78.347,Z 1135.177,A -85,B 0,C 180,E1 4624.163,E2 4624.163} C_VEL
LIN {X 0,Y 72.751,Z 1136.725,A -85,B 0,C 180,E1 4606.776,E2 4606.776} C_VEL
LIN {X 0,Y 72.131,Z 1136.963,A -85,B 0,C 180,E1 4593.553,E2 4593.553} C_VEL
LIN {X 0,Y 72.127,Z 1136.755,A -85,B 0,C 180,E1 4586.025,E2 4586.025} C_VEL
LIN {X 0,Y 72.981,Z 1135.537,A -85,B 0,C 180,E1 4571.632,E2 4571.632} C_VEL
LIN {X 0,Y 79.013,Z 1132.502,A -85,B 0,C 180,E1 4554.4,E2 4554.4} C_VEL
LIN {X 0,Y 89.213,Z 1128.456,A -85,B 0,C 180,E1 4541.329,E2 4541.329} C_VEL
LIN {X 0,Y 105.83,Z 1121.878,A -85,B 0,C 180,E1 4529.426,E2 4529.426} C_VEL
LIN {X 0,Y 122.814,Z 1114.532,A -85,B 0,C 180,E1 4521.854,E2 4521.854} C_VEL
LIN {X 0,Y 143.293,Z 1104.685,A -85,B 0,C 180,E1 4515.643,E2 4515.643} C_VEL
LIN {X 0,Y 161.321,Z 1094.818,A -85,B 0,C 180,E1 4511.675,E2 4511.675} C_VEL
LIN {X 0,Y 180.911,Z 1082.901,A -85,B 0,C 180,E1 4508.376,E2 4508.376} C_VEL
LIN {X 0,Y 200.016,Z 1069.563,A -85,B 0,C 180,E1 4505.836,E2 4505.836} C_VEL
LIN {X 0,Y 217.492,Z 1055.974,A -85,B 0,C 180,E1 4503.944,E2 4503.944} C_VEL
LIN {X 0,Y 237.147,Z 1038.626,A -85,B 0,C 180,E1 4502.181,E2 4502.181} C_VEL
LIN {X 0,Y 253.01,Z 1022.823,A -85,B 0,C 180,E1 4500.977,E2 4500.977} C_VEL
LIN {X 0,Y 270.473,Z 1003.092,A -85,B 0,C 180,E1 4499.832,E2 4499.832} C_VEL
LIN {X 0,Y 284.008,Z 985.7,A -85,B 0,C 180,E1 4499.064,E2 4499.064} C_VEL
LIN {X 0,Y 298.596,Z 964.431,A -85,B 0,C 180,E1 4498.326,E2 4498.326} C_VEL
LIN {X 0,Y 305.457,Z 953.253,A -85,B 0,C 180,E1 4498.01,E2 4498.01} C_VEL
LIN {X 0,Y 292.794,Z 973.064,A -85,B 0,C 180,E1 4497.3,E2 4497.3} C_VEL
LIN {X 0,Y 278.517,Z 992.8,A -85,B 0,C 180,E1 4496.412,E2 4496.412} C_VEL
LIN {X 0,Y 262.841,Z 1011.511,A -85,B 0,C 180,E1 4495.341,E2 4495.341} C_VEL
LIN {X 0,Y 247.266,Z 1028.071,A -85,B 0,C 180,E1 4494.141,E2 4494.141} C_VEL
LIN {X 0,Y 228.923,Z 1045.176,A -85,B 0,C 180,E1 4492.522,E2 4492.522} C_VEL
LIN {X 0,Y 212.685,Z 1058.637,A -85,B 0,C 180,E1 4490.85,E2 4490.85} C_VEL
LIN {X 0,Y 191.897,Z 1073.864,A -85,B 0,C 180,E1 4488.275,E2 4488.275} C_VEL
LIN {X 0,Y 174.451,Z 1085.097,A -85,B 0,C 180,E1 4485.616,E2 4485.616} C_VEL
LIN {X 0,Y 154.715,Z 1096.43,A -85,B 0,C 180,E1 4481.812,E2 4481.812} C_VEL
LIN {X 0,Y 135.792,Z 1105.841,A -85,B 0,C 180,E1 4476.989,E2 4476.989} C_VEL
LIN {X 0,Y 116.885,Z 1114.276,A -85,B 0,C 180,E1 4470.254,E2 4470.254} C_VEL
LIN {X 0,Y 99.986,Z 1120.807,A -85,B 0,C 180,E1 4461.263,E2 4461.263} C_VEL
LIN {X 0,Y 86.38,Z 1125.777,A -85,B 0,C 180,E1 4449.543,E2 4449.543} C_VEL
LIN {X 0,Y 76.638,Z 1129.289,A -85,B 0,C 180,E1 4433.857,E2 4433.857} C_VEL
LIN {X 0,Y 72.885,Z 1131.001,A -85,B 0,C 180,E1 4419.476,E2 4419.476} C_VEL
LIN {X 0,Y 72.193,Z 1131.693,A -85,B 0,C 180,E1 4408.413,E2 4408.413} C_VEL
LIN {X 0,Y 72.688,Z 1131.909,A -85,B 0,C 180,E1 4396.476,E2 4396.476} C_VEL
LIN {X 0,Y 76.386,Z 1131.25,A -85,B 0,C 180,E1 4381.031,E2 4381.031} C_VEL
LIN {X 0,Y 84.693,Z 1129.446,A -85,B 0,C 180,E1 4366.784,E2 4366.784} C_VEL
LIN {X 0,Y 100.164,Z 1125.498,A -85,B 0,C 180,E1 4353.014,E2 4353.014} C_VEL
LIN {X 0,Y 116.389,Z 1120.621,A -85,B 0,C 180,E1 4344.405,E2 4344.405} C_VEL
LIN {X 0,Y 137.079,Z 1113.317,A -85,B 0,C 180,E1 4337.146,E2 4337.146} C_VEL
LIN {X 0,Y 155.693,Z 1105.577,A -85,B 0,C 180,E1 4332.531,E2 4332.531} C_VEL
LIN {X 0,Y 176.962,Z 1095.411,A -85,B 0,C 180,E1 4328.58,E2 4328.58} C_VEL
LIN {X 0,Y 195.993,Z 1084.822,A -85,B 0,C 180,E1 4325.828,E2 4325.828} C_VEL
LIN {X 0,Y 216.554,Z 1071.924,A -85,B 0,C 180,E1 4323.441,E2 4323.441} C_VEL
LIN {X 0,Y 236.064,Z 1057.702,A -85,B 0,C 180,E1 4321.569,E2 4321.569} C_VEL
LIN {X 0,Y 253.974,Z 1043.064,A -85,B 0,C 180,E1 4320.118,E2 4320.118} C_VEL
LIN {X 0,Y 266.624,Z 1031.525,A -85,B 0,C 180,E1 4319.195,E2 4319.195} C_VEL
LIN {X 0,Y 249.119,Z 1047.414,A -85,B 0,C 180,E1 4318.044,E2 4318.044} C_VEL
LIN {X 0,Y 230.385,Z 1062.64,A -85,B 0,C 180,E1 4316.585,E2 4316.585} C_VEL
LIN {X 0,Y 209.891,Z 1077.117,A -85,B 0,C 180,E1 4314.656,E2 4314.656} C_VEL
LIN {X 0,Y 190.65,Z 1089.194,A -85,B 0,C 180,E1 4312.411,E2 4312.411} C_VEL
LIN {X 0,Y 168.98,Z 1101.019,A -85,B 0,C 180,E1 4309.192,E2 4309.192} C_VEL
LIN {X 0,Y 149.797,Z 1110.204,A -85,B 0,C 180,E1 4305.438,E2 4305.438} C_VEL
LIN {X 0,Y 144.165,Z 1112.705,A -85,B 0,C 180,E1 4304.112,E2 4304.112} C_VEL
LIN {X 0,Y 137.496,Z 1115.307,A -85,B 0,C 180,E1 4302.873,E2 4302.873} C_VEL
LIN {X 0,Y 118.061,Z 1121.764,A -85,B 0,C 180,E1 4300.337,E2 4300.337} C_VEL
LIN {X 0,Y 112.447,Z 1123.486,A -85,B 0,C 180,E1 4298.786,E2 4298.786} C_VEL
LIN {X 0,Y 95.213,Z 1128.761,A -85,B 0,C 180,E1 4290.649,E2 4290.649} C_VEL
LIN {X 0,Y 78.703,Z 1133.194,A -85,B 0,C 180,E1 4277.466,E2 4277.466} C_VEL
LIN {X 0,Y 68.307,Z 1135.63,A -85,B 0,C 180,E1 4260.82,E2 4260.82} C_VEL
LIN {X 0,Y 64.433,Z 1136.59,A -85,B 0,C 180,E1 4244.377,E2 4244.377} C_VEL
LIN {X 0,Y 64.173,Z 1136.625,A -85,B 0,C 180,E1 4231.786,E2 4231.786} C_VEL
LIN {X 0,Y 64.102,Z 1136.334,A -85,B 0,C 180,E1 4222.831,E2 4222.831} C_VEL
LIN {X 0,Y 66.551,Z 1134.527,A -85,B 0,C 180,E1 4204.17,E2 4204.17} C_VEL
LIN {X 0,Y 73.866,Z 1131.67,A -85,B 0,C 180,E1 4188.448,E2 4188.448} C_VEL
LIN {X 0,Y 87.972,Z 1126.769,A -85,B 0,C 180,E1 4173.844,E2 4173.844} C_VEL
LIN {X 0,Y 105.016,Z 1120.317,A -85,B 0,C 180,E1 4163.929,E2 4163.929} C_VEL
LIN {X 0,Y 124.294,Z 1112.333,A -85,B 0,C 180,E1 4156.802,E2 4156.802} C_VEL
LIN {X 0,Y 144.941,Z 1102.402,A -85,B 0,C 180,E1 4151.591,E2 4151.591} C_VEL
LIN {X 0,Y 164.577,Z 1091.77,A -85,B 0,C 180,E1 4147.98,E2 4147.98} C_VEL
LIN {X 0,Y 184.723,Z 1079.247,A -85,B 0,C 180,E1 4145.139,E2 4145.139} C_VEL
LIN {X 0,Y 202.82,Z 1066.583,A -85,B 0,C 180,E1 4143.109,E2 4143.109} C_VEL
LIN {X 0,Y 224.024,Z 1049.698,A -85,B 0,C 180,E1 4141.178,E2 4141.178} C_VEL
LIN {X 0,Y 240.975,Z 1034.365,A -85,B 0,C 180,E1 4139.906,E2 4139.906} C_VEL
LIN {X 0,Y 259.538,Z 1015.293,A -85,B 0,C 180,E1 4138.718,E2 4138.718} C_VEL
LIN {X 0,Y 273.648,Z 998.835,A -85,B 0,C 180,E1 4137.941,E2 4137.941} C_VEL
LIN {X 0,Y 274.851,Z 997.363,A -85,B 0,C 180,E1 4137.872,E2 4137.872} C_VEL
LIN {X 0,Y 260.339,Z 1014.22,A -85,B 0,C 180,E1 4136.962,E2 4136.962} C_VEL
LIN {X 0,Y 242.654,Z 1032.377,A -85,B 0,C 180,E1 4135.711,E2 4135.711} C_VEL
LIN {X 0,Y 226.069,Z 1047.305,A -85,B 0,C 180,E1 4134.365,E2 4134.365} C_VEL
LIN {X 0,Y 207.701,Z 1062.112,A -85,B 0,C 180,E1 4132.615,E2 4132.615} C_VEL
LIN {X 0,Y 188.602,Z 1075.478,A -85,B 0,C 180,E1 4130.436,E2 4130.436} C_VEL
LIN {X 0,Y 169.823,Z 1087.191,A -85,B 0,C 180,E1 4127.793,E2 4127.793} C_VEL
LIN {X 0,Y 148.761,Z 1098.605,A -85,B 0,C 180,E1 4123.981,E2 4123.981} C_VEL
LIN {X 0,Y 130.233,Z 1107.399,A -85,B 0,C 180,E1 4119.502,E2 4119.502} C_VEL
LIN {X 0,Y 109.476,Z 1115.952,A -85,B 0,C 180,E1 4112.368,E2 4112.368} C_VEL
LIN {X 0,Y 93.096,Z 1121.856,A -85,B 0,C 180,E1 4103.791,E2 4103.791} C_VEL
LIN {X 0,Y 77.062,Z 1127.107,A -85,B 0,C 180,E1 4089.478,E2 4089.478} C_VEL
LIN {X 0,Y 68.392,Z 1129.924,A -85,B 0,C 180,E1 4074.165,E2 4074.165} C_VEL
LIN {X 0,Y 64.682,Z 1131.496,A -85,B 0,C 180,E1 4057.997,E2 4057.997} C_VEL
LIN {X 0,Y 64.19,Z 1132.03,A -85,B 0,C 180,E1 4046.428,E2 4046.428} C_VEL
LIN {X 0,Y 64.962,Z 1132.174,A -85,B 0,C 180,E1 4033.915,E2 4033.915} C_VEL
LIN {X 0,Y 69.335,Z 1131.527,A -85,B 0,C 180,E1 4017.752,E2 4017.752} C_VEL
LIN {X 0,Y 78.88,Z 1129.714,A -85,B 0,C 180,E1 4002.675,E2 4002.675} C_VEL
LIN {X 0,Y 95.894,Z 1125.748,A -85,B 0,C 180,E1 3988.851,E2 3988.851} C_VEL
LIN {X 0,Y 112.591,Z 1121.044,A -85,B 0,C 180,E1 3980.808,E2 3980.808} C_VEL
LIN {X 0,Y 133.965,Z 1113.881,A -85,B 0,C 180,E1 3973.999,E2 3973.999} C_VEL
LIN {X 0,Y 153.17,Z 1106.182,A -85,B 0,C 180,E1 3969.69,E2 3969.69} C_VEL
LIN {X 0,Y 173.995,Z 1096.604,A -85,B 0,C 180,E1 3966.186,E2 3966.186} C_VEL
LIN {X 0,Y 194.347,Z 1085.559,A -85,B 0,C 180,E1 3963.522,E2 3963.522} C_VEL
LIN {X 0,Y 214.047,Z 1073.464,A -85,B 0,C 180,E1 3961.455,E2 3961.455} C_VEL
LIN {X 0,Y 233.978,Z 1059.36,A -85,B 0,C 180,E1 3959.724,E2 3959.724} C_VEL
LIN {X 0,Y 239.306,Z 1055.291,A -85,B 0,C 180,E1 3959.295,E2 3959.295} C_VEL
LIN {X 0,Y 221.032,Z 1068.977,A -85,B 0,C 180,E1 3957.926,E2 3957.926} C_VEL
LIN {X 0,Y 199.479,Z 1083.224,A -85,B 0,C 180,E1 3955.945,E2 3955.945} C_VEL
LIN {X 0,Y 180.065,Z 1094.367,A -85,B 0,C 180,E1 3953.71,E2 3953.71} C_VEL
LIN {X 0,Y 158.179,Z 1105.453,A -85,B 0,C 180,E1 3950.442,E2 3950.442} C_VEL
LIN {X 0,Y 136.964,Z 1114.536,A -85,B 0,C 180,E1 3946.157,E2 3946.157} C_VEL
LIN {X 0,Y 115.936,Z 1122.388,A -85,B 0,C 180,E1 3940.064,E2 3940.064} C_VEL
LIN {X 0,Y 112.447,Z 1123.486,A -85,B 0,C 180,E1 3938.786,E2 3938.786} C_VEL
LIN {X 0,Y 105.906,Z 1125.433,A -85,B 0,C 180,E1 3936.818,E2 3936.818} C_VEL
LIN {X 0,Y 86.806,Z 1129.904,A -85,B 0,C 180,E1 3931.922,E2 3931.922} C_VEL
LIN {X 0,Y 81.625,Z 1130.98,A -85,B 0,C 180,E1 3929.183,E2 3929.183} C_VEL
LIN {X 0,Y 67.477,Z 1134.151,A -85,B 0,C 180,E1 3915.339,E2 3915.339} C_VEL
LIN {X 0,Y 57.776,Z 1136.095,A -85,B 0,C 180,E1 3893.456,E2 3893.456} C_VEL
LIN {X 0,Y 56.115,Z 1136.392,A -85,B 0,C 180,E1 3875.111,E2 3875.111} C_VEL
LIN {X 0,Y 56.151,Z 1136.224,A -85,B 0,C 180,E1 3866.938,E2 3866.938} C_VEL
LIN {X 0,Y 57.163,Z 1135.152,A -85,B 0,C 180,E1 3849.522,E2 3849.522} C_VEL
LIN {X 0,Y 65.31,Z 1132.186,A -85,B 0,C 180,E1 3827.651,E2 3827.651} C_VEL
LIN {X 0,Y 77.872,Z 1128.212,A -85,B 0,C 180,E1 3813.424,E2 3813.424} C_VEL
LIN {X 0,Y 96.101,Z 1122.158,A -85,B 0,C 180,E1 3802.178,E2 3802.178} C_VEL
LIN {X 0,Y 115.849,Z 1114.518,A -85,B 0,C 180,E1 3794.833,E2 3794.833} C_VEL
LIN {X 0,Y 136.912,Z 1105.304,A -85,B 0,C 180,E1 3789.621,E2 3789.621} C_VEL
LIN {X 0,Y 157.829,Z 1094.533,A -85,B 0,C 180,E1 3785.933,E2 3785.933} C_VEL
LIN {X 0,Y 178.425,Z 1082.555,A -85,B 0,C 180,E1 3783.213,E2 3783.213} C_VEL
LIN {X 0,Y 199.015,Z 1068.673,A -85,B 0,C 180,E1 3781.085,E2 3781.085} C_VEL
LIN {X 0,Y 217.985,Z 1054.269,A -85,B 0,C 180,E1 3779.509,E2 3779.509} C_VEL
LIN {X 0,Y 237.093,Z 1037.642,A -85,B 0,C 180,E1 3778.196,E2 3778.196} C_VEL
LIN {X 0,Y 244.363,Z 1030.854,A -85,B 0,C 180,E1 3777.756,E2 3777.756} C_VEL
LIN {X 0,Y 226.403,Z 1046.942,A -85,B 0,C 180,E1 3776.483,E2 3776.483} C_VEL
LIN {X 0,Y 207.792,Z 1061.81,A -85,B 0,C 180,E1 3774.927,E2 3774.927} C_VEL
LIN {X 0,Y 187.427,Z 1075.902,A -85,B 0,C 180,E1 3772.878,E2 3772.878} C_VEL
LIN {X 0,Y 168.295,Z 1087.602,A -85,B 0,C 180,E1 3770.491,E2 3770.491} C_VEL
LIN {X 0,Y 146.453,Z 1099.125,A -85,B 0,C 180,E1 3766.979,E2 3766.979} C_VEL
LIN {X 0,Y 127.616,Z 1107.775,A -85,B 0,C 180,E1 3762.92,E2 3762.92} C_VEL
LIN {X 0,Y 105.955,Z 1116.306,A -85,B 0,C 180,E1 3756.261,E2 3756.261} C_VEL
LIN {X 0,Y 89.206,Z 1121.984,A -85,B 0,C 180,E1 3748.416,E2 3748.416} C_VEL
LIN {X 0,Y 72.182,Z 1127.124,A -85,B 0,C 180,E1 3734.949,E2 3734.949} C_VEL
LIN {X 0,Y 61.501,Z 1130.127,A -85,B 0,C 180,E1 3718.131,E2 3718.131} C_VEL
LIN {X 0,Y 56.878,Z 1131.731,A -85,B 0,C 180,E1 3700.111,E2 3700.111} C_VEL
LIN {X 0,Y 56.193,Z 1132.296,A -85,B 0,C 180,E1 3686.94,E2 3686.94} C_VEL
LIN {X 0,Y 57.072,Z 1132.476,A -85,B 0,C 180,E1 3672.672,E2 3672.672} C_VEL
LIN {X 0,Y 62.554,Z 1131.804,A -85,B 0,C 180,E1 3653.742,E2 3653.742} C_VEL
LIN {X 0,Y 73.537,Z 1129.983,A -85,B 0,C 180,E1 3637.942,E2 3637.942} C_VEL
LIN {X 0,Y 92.176,Z 1125.998,A -85,B 0,C 180,E1 3624.328,E2 3624.328} C_VEL
LIN {X 0,Y 109.686,Z 1121.348,A -85,B 0,C 180,E1 3616.827,E2 3616.827} C_VEL
LIN {X 0,Y 132.199,Z 1114.1,A -85,B 0,C 180,E1 3610.496,E2 3610.496} C_VEL
LIN {X 0,Y 151.991,Z 1106.389,A -85,B 0,C 180,E1 3606.599,E2 3606.599} C_VEL
LIN {X 0,Y 173.297,Z 1096.791,A -85,B 0,C 180,E1 3603.456,E2 3603.456} C_VEL
LIN {X 0,Y 194.014,Z 1085.728,A -85,B 0,C 180,E1 3601.08,E2 3601.08} C_VEL
LIN {X 0,Y 211.99,Z 1074.88,A -85,B 0,C 180,E1 3599.391,E2 3599.391} C_VEL
LIN {X 0,Y 193.127,Z 1086.532,A -85,B 0,C 180,E1 3597.762,E2 3597.762} C_VEL
LIN {X 0,Y 170.559,Z 1098.761,A -85,B 0,C 180,E1 3595.286,E2 3595.286} C_VEL
LIN {X 0,Y 150.171,Z 1108.198,A -85,B 0,C 180,E1 3592.347,E2 3592.347} C_VEL
LIN {X 0,Y 128.735,Z 1116.847,A -85,B 0,C 180,E1 3588.141,E2 3588.141} C_VEL
LIN {X 0,Y 107.249,Z 1123.992,A -85,B 0,C 180,E1 3581.981,E2 3581.981} C_VEL
LIN {X 0,Y 88.301,Z 1129.373,A -85,B 0,C 180,E1 3573.453,E2 3573.453} C_VEL
LIN {X 0,Y 81.625,Z 1130.98,A -85,B 0,C 180,E1 3569.183,E2 3569.183} C_VEL
LIN {X 0,Y 75.734,Z 1132.249,A -85,B 0,C 180,E1 3565.601,E2 3565.601} C_VEL
LIN {X 0,Y 58.282,Z 1134.676,A -85,B 0,C 180,E1 3554.472,E2 3554.472} C_VEL
LIN {X 0,Y 54.775,Z 1135.093,A -85,B 0,C 180,E1 3549.403,E2 3549.403} C_VEL
LIN {X 0,Y 48.592,Z 1136.081,A -85,B 0,C 180,E1 3526.743,E2 3526.743} C_VEL
LIN {X 0,Y 48.189,Z 1136.026,A -85,B 0,C 180,E1 3511.189,E2 3511.189} C_VEL
LIN {X 0,Y 48.223,Z 1135.586,A -85,B 0,C 180,E1 3498.033,E2 3498.033} C_VEL
LIN {X 0,Y 52.687,Z 1133.776,A -85,B 0,C 180,E1 3475.296,E2 3475.296} C_VEL
LIN {X 0,Y 63.767,Z 1130.677,A -85,B 0,C 180,E1 3456.899,E2 3456.899} C_VEL
LIN {X 0,Y 83.124,Z 1125.029,A -85,B 0,C 180,E1 3442.146,E2 3442.146} C_VEL
LIN {X 0,Y 101.229,Z 1118.966,A -85,B 0,C 180,E1 3434.533,E2 3434.533} C_VEL
LIN {X 0,Y 123.367,Z 1110.357,A -85,B 0,C 180,E1 3428.576,E2 3428.576} C_VEL
LIN {X 0,Y 143.503,Z 1101.141,A -85,B 0,C 180,E1 3424.871,E2 3424.871} C_VEL
LIN {X 0,Y 165.078,Z 1089.868,A -85,B 0,C 180,E1 3421.95,E2 3421.95} C_VEL
LIN {X 0,Y 185.982,Z 1077.083,A -85,B 0,C 180,E1 3419.796,E2 3419.796} C_VEL
LIN {X 0,Y 206.084,Z 1063.217,A -85,B 0,C 180,E1 3418.165,E2 3418.165} C_VEL
LIN {X 0,Y 213.484,Z 1057.481,A -85,B 0,C 180,E1 3417.647,E2 3417.647} C_VEL
LIN {X 0,Y 194.435,Z 1071.251,A -85,B 0,C 180,E1 3416.08,E2 3416.08} C_VEL
LIN {X 0,Y 173.926,Z 1084.089,A -85,B 0,C 180,E1 3414.027,E2 3414.027} C_VEL
LIN {X 0,Y 154.645,Z 1094.678,A -85,B 0,C 180,E1 3411.594,E2 3411.594} C_VEL
LIN {X 0,Y 131.361,Z 1105.647,A -85,B 0,C 180,E1 3407.694,E2 3407.694} C_VEL
LIN {X 0,Y 111.819,Z 1113.493,A -85,B 0,C 180,E1 3403.098,E2 3403.098} C_VEL
LIN {X 0,Y 89.324,Z 1121.101,A -85,B 0,C 180,E1 3395.056,E2 3395.056} C_VEL
LIN {X 0,Y 72.947,Z 1125.781,A -85,B 0,C 180,E1 3385.328,E2 3385.328} C_VEL
LIN {X 0,Y 57.32,Z 1129.792,A -85,B 0,C 180,E1 3367.629,E2 3367.629} C_VEL
LIN {X 0,Y 49.727,Z 1131.772,A -85,B 0,C 180,E1 3346.35,E2 3346.35} C_VEL
LIN {X 0,Y 48.209,Z 1132.539,A -85,B 0,C 180,E1 3328.812,E2 3328.812} C_VEL
LIN {X 0,Y 49.056,Z 1132.795,A -85,B 0,C 180,E1 3312.197,E2 3312.197} C_VEL
LIN {X 0,Y 55.673,Z 1132.142,A -85,B 0,C 180,E1 3289.716,E2 3289.716} C_VEL
LIN {X 0,Y 68.072,Z 1130.358,A -85,B 0,C 180,E1 3273.148,E2 3273.148} C_VEL
LIN {X 0,Y 88.235,Z 1126.447,A -85,B 0,C 180,E1 3259.853,E2 3259.853} C_VEL
LIN {X 0,Y 107.573,Z 1121.588,A -85,B 0,C 180,E1 3252.582,E2 3252.582} C_VEL
LIN {X 0,Y 130.939,Z 1114.318,A -85,B 0,C 180,E1 3246.914,E2 3246.914} C_VEL
LIN {X 0,Y 151.261,Z 1106.596,A -85,B 0,C 180,E1 3243.469,E2 3243.469} C_VEL
LIN {X 0,Y 173.991,Z 1096.467,A -85,B 0,C 180,E1 3240.6,E2 3240.6} C_VEL
LIN {X 0,Y 184.616,Z 1091.062,A -85,B 0,C 180,E1 3239.502,E2 3239.502} C_VEL
LIN {X 0,Y 164.151,Z 1101.364,A -85,B 0,C 180,E1 3237.407,E2 3237.407} C_VEL
LIN {X 0,Y 141.43,Z 1111.296,A -85,B 0,C 180,E1 3234.32,E2 3234.32} C_VEL
LIN {X 0,Y 119.74,Z 1119.136,A -85,B 0,C 180,E1 3230.186,E2 3230.186} C_VEL
LIN {X 0,Y 97.816,Z 1125.857,A -85,B 0,C 180,E1 3223.923,E2 3223.923} C_VEL
LIN {X 0,Y 77.626,Z 1130.738,A -85,B 0,C 180,E1 3214.378,E2 3214.378} C_VEL
LIN {X 0,Y 61.967,Z 1133.882,A -85,B 0,C 180,E1 3200.762,E2 3200.762} C_VEL
LIN {X 0,Y 54.775,Z 1135.093,A -85,B 0,C 180,E1 3189.403,E2 3189.403} C_VEL
LIN {X 0,Y 50.648,Z 1135.668,A -85,B 0,C 180,E1 3181.56,E2 3181.56} C_VEL
LIN {X 0,Y 44.122,Z 1135.931,A -85,B 0,C 180,E1 3168.083,E2 3168.083} C_VEL
LIN {X 0,Y 40.187,Z 1135.695,A -85,B 0,C 180,E1 3148.733,E2 3148.733} C_VEL
LIN {X 0,Y 41.05,Z 1134.915,A -85,B 0,C 180,E1 3128.57,E2 3128.57} C_VEL
LIN {X 0,Y 48.776,Z 1132.852,A -85,B 0,C 180,E1 3104.152,E2 3104.152} C_VEL
LIN {X 0,Y 66.867,Z 1128.4,A -85,B 0,C 180,E1 3084.193,E2 3084.193} C_VEL
LIN {X 0,Y 84.799,Z 1123.353,A -85,B 0,C 180,E1 3074.784,E2 3074.784} C_VEL
LIN {X 0,Y 107.963,Z 1115.6,A -85,B 0,C 180,E1 3067.703,E2 3067.703} C_VEL
LIN {X 0,Y 128.256,Z 1107.469,A -85,B 0,C 180,E1 3063.714,E2 3063.714} C_VEL
LIN {X 0,Y 150.991,Z 1096.889,A -85,B 0,C 180,E1 3060.558,E2 3060.558} C_VEL
LIN {X 0,Y 172.049,Z 1085.337,A -85,B 0,C 180,E1 3058.407,E2 3058.407} C_VEL
LIN {X 0,Y 182.48,Z 1079.035,A -85,B 0,C 180,E1 3057.532,E2 3057.532} C_VEL
LIN {X 0,Y 159.526,Z 1092.062,A -85,B 0,C 180,E1 3055.274,E2 3055.274} C_VEL
LIN {X 0,Y 140.092,Z 1101.556,A -85,B 0,C 180,E1 3052.795,E2 3052.795} C_VEL
LIN {X 0,Y 115.955,Z 1111.573,A -85,B 0,C 180,E1 3048.561,E2 3048.561} C_VEL
LIN {X 0,Y 95.989,Z 1118.48,A -85,B 0,C 180,E1 3043.405,E2 3043.405} C_VEL
LIN {X 0,Y 73.491,Z 1124.924,A -85,B 0,C 180,E1 3033.893,E2 3033.893} C_VEL
LIN {X 0,Y 56.956,Z 1128.812,A -85,B 0,C 180,E1 3020.802,E2 3020.802} C_VEL
LIN {X 0,Y 44.34,Z 1131.612,A -85,B 0,C 180,E1 2998.266,E2 2998.266} C_VEL
LIN {X 0,Y 40.321,Z 1132.761,A -85,B 0,C 180,E1 2972.843,E2 2972.843} C_VEL
LIN {X 0,Y 40.754,Z 1133.08,A -85,B 0,C 180,E1 2954.343,E2 2954.343} C_VEL
LIN {X 0,Y 48.075,Z 1132.603,A -85,B 0,C 180,E1 2926.657,E2 2926.657} C_VEL
LIN {X 0,Y 61.649,Z 1130.945,A -85,B 0,C 180,E1 2908.856,E2 2908.856} C_VEL
LIN {X 0,Y 81.344,Z 1127.672,A -85,B 0,C 180,E1 2896.506,E2 2896.506} C_VEL
LIN {X 0,Y 103.323,Z 1122.546,A -85,B 0,C 180,E1 2888.908,E2 2888.908} C_VEL
LIN {X 0,Y 125.327,Z 1116.189,A -85,B 0,C 180,E1 2884.118,E2 2884.118} C_VEL
LIN {X 0,Y 147.995,Z 1107.998,A -85,B 0,C 180,E1 2880.693,E2 2880.693} C_VEL
LIN {X 0,Y 156.988,Z 1104.415,A -85,B 0,C 180,E1 2879.59,E2 2879.59} C_VEL
LIN {X 0,Y 134.202,Z 1113.516,A -85,B 0,C 180,E1 2876.749,E2 2876.749} C_VEL
LIN {X 0,Y 110.922,Z 1121.395,A -85,B 0,C 180,E1 2872.563,E2 2872.563} C_VEL
LIN {X 0,Y 88.501,Z 1127.365,A -85,B 0,C 180,E1 2866.275,E2 2866.275} C_VEL
LIN {X 0,Y 68.593,Z 1131.661,A -85,B 0,C 180,E1 2856.689,E2 2856.689} C_VEL
LIN {X 0,Y 50.57,Z 1134.568,A -85,B 0,C 180,E1 2838.707,E2 2838.707} C_VEL
LIN {X 0,Y 41.755,Z 1135.676,A -85,B 0,C 180,E1 2815.534,E2 2815.534} C_VEL
LIN {X 0,Y 40.133,Z 1135.774,A -85,B 0,C 180,E1 2794.286,E2 2794.286} C_VEL
LIN {X 0,Y 40.187,Z 1135.695,A -85,B 0,C 180,E1 2788.733,E2 2788.733} C_VEL
LIN {X 0,Y 39.572,Z 1135.453,A -85,B 0,C 180,E1 2779.269,E2 2779.269} C_VEL
LIN {X 0,Y 38.277,Z 1134.768,A -85,B 0,C 180,E1 2765.436,E2 2765.436} C_VEL
LIN {X 0,Y 39.71,Z 1133.395,A -85,B 0,C 180,E1 2744.682,E2 2744.682} C_VEL
LIN {X 0,Y 42.496,Z 1132.713,A -85,B 0,C 180,E1 2737.891,E2 2737.891} C_VEL
LIN {X 0,Y 62.183,Z 1128.494,A -85,B 0,C 180,E1 2718.428,E2 2718.428} C_VEL
LIN {X 0,Y 82.127,Z 1123.268,A -85,B 0,C 180,E1 2709.54,E2 2709.54} C_VEL
LIN {X 0,Y 105.205,Z 1115.958,A -85,B 0,C 180,E1 2703.67,E2 2703.67} C_VEL
LIN {X 0,Y 126.987,Z 1107.503,A -85,B 0,C 180,E1 2700.125,E2 2700.125} C_VEL
LIN {X 0,Y 149.115,Z 1097.519,A -85,B 0,C 180,E1 2697.598,E2 2697.598} C_VEL
LIN {X 0,Y 150.973,Z 1096.566,A -85,B 0,C 180,E1 2697.395,E2 2697.395} C_VEL
LIN {X 0,Y 128.532,Z 1106.539,A -85,B 0,C 180,E1 2694.718,E2 2694.718} C_VEL
LIN {X 0,Y 107.261,Z 1114.565,A -85,B 0,C 180,E1 2691.166,E2 2691.166} C_VEL
LIN {X 0,Y 83.781,Z 1121.787,A -85,B 0,C 180,E1 2685.172,E2 2685.172} C_VEL
LIN {X 0,Y 64.259,Z 1126.644,A -85,B 0,C 180,E1 2676.645,E2 2676.645} C_VEL
LIN {X 0,Y 44.29,Z 1130.629,A -85,B 0,C 180,E1 2658.16,E2 2658.16} C_VEL
LIN {X 0,Y 34.634,Z 1132.371,A -85,B 0,C 180,E1 2633.84,E2 2633.84} C_VEL
LIN {X 0,Y 32.232,Z 1133.095,A -85,B 0,C 180,E1 2610,E2 2610} C_VEL
LIN {X 0,Y 33.461,Z 1133.397,A -85,B 0,C 180,E1 2587.141,E2 2587.141} C_VEL
LIN {X 0,Y 43.769,Z 1132.758,A -85,B 0,C 180,E1 2556.911,E2 2556.911} C_VEL
LIN {X 0,Y 59.789,Z 1131.003,A -85,B 0,C 180,E1 2540.523,E2 2540.523} C_VEL
LIN {X 0,Y 83.122,Z 1127.146,A -85,B 0,C 180,E1 2529.459,E2 2529.459} C_VEL
LIN {X 0,Y 104.232,Z 1122.315,A -85,B 0,C 180,E1 2523.911,E2 2523.911} C_VEL
LIN {X 0,Y 127.987,Z 1115.447,A -85,B 0,C 180,E1 2519.887,E2 2519.887} C_VEL
LIN {X 0,Y 129.245,Z 1115.012,A -85,B 0,C 180,E1 2519.713,E2 2519.713} C_VEL
LIN {X 0,Y 104.276,Z 1122.744,A -85,B 0,C 180,E1 2515.748,E2 2515.748} C_VEL
LIN {X 0,Y 83.144,Z 1127.974,A -85,B 0,C 180,E1 2510.45,E2 2510.45} C_VEL
LIN {X 0,Y 59.692,Z 1132.361,A -85,B 0,C 180,E1 2499.727,E2 2499.727} C_VEL
LIN {X 0,Y 42.856,Z 1134.597,A -85,B 0,C 180,E1 2482.493,E2 2482.493} C_VEL
LIN {X 0,Y 32.723,Z 1135.6,A -85,B 0,C 180,E1 2449.641,E2 2449.641} C_VEL
LIN {X 0,Y 32.192,Z 1135.416,A -85,B 0,C 180,E1 2429.196,E2 2429.196} C_VEL
LIN {X 0,Y 33.345,Z 1134.686,A -85,B 0,C 180,E1 2405.177,E2 2405.177} C_VEL
LIN {X 0,Y 42.496,Z 1132.713,A -85,B 0,C 180,E1 2377.891,E2 2377.891} C_VEL
LIN {X 0,Y 46.93,Z 1131.722,A -85,B 0,C 180,E1 2369.813,E2 2369.813} C_VEL
LIN {X 0,Y 60.256,Z 1128.186,A -85,B 0,C 180,E1 2351.496,E2 2351.496} C_VEL
LIN {X 0,Y 65.388,Z 1126.931,A -85,B 0,C 180,E1 2348.658,E2 2348.658} C_VEL
LIN {X 0,Y 89.153,Z 1120.678,A -85,B 0,C 180,E1 2341.928,E2 2341.928} C_VEL
LIN {X 0,Y 111.039,Z 1113.394,A -85,B 0,C 180,E1 2338.273,E2 2338.273} C_VEL
LIN {X 0,Y 118.763,Z 1110.594,A -85,B 0,C 180,E1 2337.243,E2 2337.243} C_VEL
LIN {X 0,Y 95.577,Z 1118.308,A -85,B 0,C 180,E1 2333.647,E2 2333.647} C_VEL
LIN {X 0,Y 72.606,Z 1124.583,A -85,B 0,C 180,E1 2327.898,E2 2327.898} C_VEL
LIN {X 0,Y 50.837,Z 1129.02,A -85,B 0,C 180,E1 2317.583,E2 2317.583} C_VEL
LIN {X 0,Y 34.322,Z 1131.693,A -85,B 0,C 180,E1 2299.241,E2 2299.241} C_VEL
LIN {X 0,Y 24.732,Z 1133.254,A -85,B 0,C 180,E1 2261.663,E2 2261.663} C_VEL
LIN {X 0,Y 24.515,Z 1133.531,A -85,B 0,C 180,E1 2235.834,E2 2235.834} C_VEL
LIN {X 0,Y 31.004,Z 1133.512,A -85,B 0,C 180,E1 2202.118,E2 2202.118} C_VEL
LIN {X 0,Y 49.608,Z 1132.195,A -85,B 0,C 180,E1 2177.598,E2 2177.598} C_VEL
LIN {X 0,Y 70.545,Z 1129.406,A -85,B 0,C 180,E1 2167.172,E2 2167.172} C_VEL
LIN {X 0,Y 94.008,Z 1125.009,A -85,B 0,C 180,E1 2161.106,E2 2161.106} C_VEL
LIN {X 0,Y 100.895,Z 1123.318,A -85,B 0,C 180,E1 2159.843,E2 2159.843} C_VEL
LIN {X 0,Y 76.326,Z 1128.943,A -85,B 0,C 180,E1 2154.637,E2 2154.637} C_VEL
LIN {X 0,Y 54.613,Z 1132.46,A -85,B 0,C 180,E1 2146.018,E2 2146.018} C_VEL
LIN {X 0,Y 35.402,Z 1134.627,A -85,B 0,C 180,E1 2127.92,E2 2127.92} C_VEL
LIN {X 0,Y 24.401,Z 1135.259,A -85,B 0,C 180,E1 2086.669,E2 2086.669} C_VEL
LIN {X 0,Y 24.162,Z 1135.113,A -85,B 0,C 180,E1 2067.628,E2 2067.628} C_VEL
LIN {X 0,Y 27.442,Z 1134.158,A -85,B 0,C 180,E1 2031.726,E2 2031.726} C_VEL
LIN {X 0,Y 44.21,Z 1131.345,A -85,B 0,C 180,E1 2001.215,E2 2001.215} C_VEL
LIN {X 0,Y 63.828,Z 1127.288,A -85,B 0,C 180,E1 1989.275,E2 1989.275} C_VEL
LIN {X 0,Y 65.388,Z 1126.931,A -85,B 0,C 180,E1 1988.658,E2 1988.658} C_VEL
LIN {X 0,Y 69.63,Z 1125.903,A -85,B 0,C 180,E1 1986.221,E2 1986.221} C_VEL
LIN {X 0,Y 79.824,Z 1122.925,A -85,B 0,C 180,E1 1978.648,E2 1978.648} C_VEL
LIN {X 0,Y 83.814,Z 1121.841,A -85,B 0,C 180,E1 1977.41,E2 1977.41} C_VEL
LIN {X 0,Y 85.499,Z 1121.396,A -85,B 0,C 180,E1 1977.073,E2 1977.073} C_VEL
LIN {X 0,Y 63.573,Z 1126.516,A -85,B 0,C 180,E1 1972.257,E2 1972.257} C_VEL
LIN {X 0,Y 41.874,Z 1130.409,A -85,B 0,C 180,E1 1962.774,E2 1962.774} C_VEL
LIN {X 0,Y 22.243,Z 1132.843,A -85,B 0,C 180,E1 1935.992,E2 1935.992} C_VEL
LIN {X 0,Y 16.295,Z 1133.651,A -85,B 0,C 180,E1 1893.518,E2 1893.518} C_VEL
LIN {X 0,Y 18.566,Z 1133.959,A -85,B 0,C 180,E1 1853.671,E2 1853.671} C_VEL
LIN {X 0,Y 35.465,Z 1133.374,A -85,B 0,C 180,E1 1816.546,E2 1816.546} C_VEL
LIN {X 0,Y 55.194,Z 1131.648,A -85,B 0,C 180,E1 1804.881,E2 1804.881} C_VEL
LIN {X 0,Y 71.731,Z 1129.403,A -85,B 0,C 180,E1 1800,E2 1800} C_VEL
LIN {X 0,Y 50.319,Z 1132.56,A -85,B 0,C 180,E1 1793.49,E2 1793.49} C_VEL
LIN {X 0,Y 26.611,Z 1134.642,A -85,B 0,C 180,E1 1773.199,E2 1773.199} C_VEL
LIN {X 0,Y 16.376,Z 1134.934,A -85,B 0,C 180,E1 1727.775,E2 1727.775} C_VEL
LIN {X 0,Y 16.146,Z 1134.822,A -85,B 0,C 180,E1 1706.449,E2 1706.449} C_VEL
LIN {X 0,Y 22.998,Z 1133.704,A -85,B 0,C 180,E1 1654.304,E2 1654.304} C_VEL
LIN {X 0,Y 44.732,Z 1130.516,A -85,B 0,C 180,E1 1629.002,E2 1629.002} C_VEL
LIN {X 0,Y 65.01,Z 1126.516,A -85,B 0,C 180,E1 1621.289,E2 1621.289} C_VEL
LIN {X 0,Y 83.814,Z 1121.841,A -85,B 0,C 180,E1 1617.41,E2 1617.41} C_VEL
LIN {X 0,Y 82.027,Z 1122.308,A -85,B 0,C 180,E1 1616.758,E2 1616.758} C_VEL
LIN {X 0,Y 72.197,Z 1124.762,A -85,B 0,C 180,E1 1616.261,E2 1616.261} C_VEL
LIN {X 0,Y 50.462,Z 1129.223,A -85,B 0,C 180,E1 1617.498,E2 1617.498} C_VEL
LIN {X 0,Y 38.372,Z 1131.159,A -85,B 0,C 180,E1 1620.324,E2 1620.324} C_VEL
LIN {X 0,Y 16.02,Z 1133.698,A -85,B 0,C 180,E1 1640.567,E2 1640.567} C_VEL
LIN {X 0,Y 8.174,Z 1134.557,A -85,B 0,C 180,E1 1710,E2 1710} C_VEL
LIN {X 0,Y 17.796,Z 1134.566,A -85,B 0,C 180,E1 1782.782,E2 1782.782} C_VEL
LIN {X 0,Y 37.999,Z 1133.455,A -85,B 0,C 180,E1 1799.296,E2 1799.296} C_VEL
LIN {X 0,Y 40.695,Z 1133.246,A -85,B 0,C 180,E1 1800.285,E2 1800.285} C_VEL
LIN {X 0,Y 20.635,Z 1134.133,A -85,B 0,C 180,E1 1814.271,E2 1814.271} C_VEL
LIN {X 0,Y 8.857,Z 1134.062,A -85,B 0,C 180,E1 1863.155,E2 1863.155} C_VEL
LIN {X 0,Y 10.141,Z 1133.787,A -85,B 0,C 180,E1 1926.269,E2 1926.269} C_VEL
LIN {X 0,Y 27.691,Z 1132.207,A -85,B 0,C 180,E1 1967.147,E2 1967.147} C_VEL
LIN {X 0,Y 48.092,Z 1129.512,A -85,B 0,C 180,E1 1976.362,E2 1976.362} C_VEL
LIN {X 0,Y 49.762,Z 1129.257,A -85,B 0,C 180,E1 1976.884,E2 1976.884} C_VEL
LIN {X 0,Y 38.372,Z 1131.159,A -85,B 0,C 180,E1 1980.324,E2 1980.324} C_VEL
LIN {X 0,Y 29.557,Z 1132.326,A -85,B 0,C 180,E1 1982.559,E2 1982.559} C_VEL
LIN {X 0,Y 15.102,Z 1133.596,A -85,B 0,C 180,E1 1981.679,E2 1981.679} C_VEL
LIN {X 0,Y 1.772,Z 1134.219,A -85,B 0,C 180,E1 1970.442,E2 1970.442} C_VEL
LIN {X 0,Y 0.225,Z 1134.255,A -85,B 0,C 180,E1 1870.869,E2 1870.869} C_VEL
LIN {X 0,Y 1.5,Z 1134.292,A -85,B 0,C 180,E1 1802.117,E2 1802.117} C_VEL
LIN {X 0,Y 2.005,Z 1134.213,A -85,B 0,C 180,E1 1975.912,E2 1975.912} C_VEL
LIN {X 0,Y 2.829,Z 1134.19,A -85,B 0,C 180,E1 1974.601,E2 1974.601} C_VEL
LIN {X 0,Y 0.225,Z 1134.255,A -85,B 0,C 180,E1 1870.869,E2 1870.869} C_VEL
LIN {X 0,Y 2.024,Z 1136.255,A -85,B 0,C 180,E1 1802.55,E2 1802.55} C_VEL
LIN {X 0,Y 2.024,Z 1164.5,A -85,B 0,C 180,E1 1802.55,E2 1802.55} C_VEL
LIN {X 0,Y 2.024,Z 1164.5,A -85,B 0,C 180,E1 1802.55,E2 1802.55}

QRS_NEXT_CUT()

QRS_NEXT()
QRS_HOME()

END
